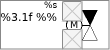
VISUALIZATION StellAntrieb_ML_Valve_Flow_LA_CheckEnabled  // 110x50
VAR_INPUT
    ITF_STELLANTRIEB_IN   	:   ITF_STELLANTRIEB;
	stExklParameter			:	STRING[40];
END_VAR
    Frame (61,0 50x50), invisible if: NOT ITF_STELLANTRIEB_IN.proIsEnabled
        shows Icon_ML_Durchfluss(ITF_STELLANTRIEB_IN := ITF_STELLANTRIEB_IN)
    Frame (0,0 60x25), invisible if: NOT ITF_STELLANTRIEB_IN.proIsEnabled
        shows ValueUpDwn(ITF_STELLANTRIEB_IN := ITF_STELLANTRIEB_IN, uiTextAusrichtung := 6)
    Rectangle (0,0 110x50)
        OnMouseClick:  Dialog=StellAntrieb_POPUP, Parameters={stExklParameter: stExklParameter, ITF_STELLANTRIEBIN: ITF_STELLANTRIEB_IN, uiPopUpGruppe: 0}, OpenCentered=True
END_VISUALIZATION

// 40 Visualizations/ICON/StellAntrieb_LEFT/Motor_LEFT/Valve_Flow/Above/StellAntrieb_ML_Valve_Flow_LA_CheckQuerry
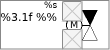
VISUALIZATION StellAntrieb_ML_Valve_Flow_LA_CheckQuerry  // 110x50
VAR_INPUT
    ITF_STELLANTRIEB_IN   	:   ITF_STELLANTRIEB;
	stExklParameter			:	STRING[40];
END_VAR
    Frame (0,0 110x50)
        shows StellAntrieb_ML_Valve_Flow_LA_CheckEnabled(ITF_STELLANTRIEB_IN := ITF_STELLANTRIEB_IN, stExklParameter := stExklParameter)
END_VISUALIZATION

// 40 Visualizations/ICON/StellAntrieb_LEFT/Motor_LEFT/Valve_Flow/Above/StellAntrieb_ML_Valve_Flow_Txt_L_Above
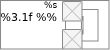
VISUALIZATION StellAntrieb_ML_Valve_Flow_Txt_L_Above  // 110x50
VAR_INPUT
    ITF_STELLANTRIEB_IN   	:   ITF_STELLANTRIEB;	
END_VAR
VAR_INPUT CONSTANT
	stExklParameter			:	STRING[40] := '';
END_VAR
VAR CONSTANT
	uiIconNr				: 	UINT := 12;
END_VAR
    Frame (0,0 110x50), invisible if: NOT fcCheckQuerryReturnIcon(_ITF_In := ITF_STELLANTRIEB_IN,_uiIconNr_In := uiIconNr)
        shows StellAntrieb_ML_Valve_Flow_LA_CheckQuerry(ITF_STELLANTRIEB_IN := ITF_STELLANTRIEB_IN, stExklParameter := stExklParameter)
        shows S_AT_ML_Valve_AB_Up_LA_CheckQuerry()
END_VISUALIZATION

// 40 Visualizations/ICON/StellAntrieb_LEFT/Motor_LEFT/Valve_Flow/Below/StellAntrieb_ML_Valve_Flow_LB_CheckEnabled
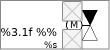
VISUALIZATION StellAntrieb_ML_Valve_Flow_LB_CheckEnabled  // 110x50
VAR_INPUT
    ITF_STELLANTRIEB_IN   	:   ITF_STELLANTRIEB;	
	stExklParameter			:	STRING[40];
END_VAR
    Frame (61,0 50x50), invisible if: NOT ITF_STELLANTRIEB_IN.proIsEnabled
        shows Icon_ML_Durchfluss(ITF_STELLANTRIEB_IN := ITF_STELLANTRIEB_IN)
    Frame (0,25 60x25), invisible if: NOT ITF_STELLANTRIEB_IN.proIsEnabled
        shows ValueDwnUp(ITF_STELLANTRIEB_IN := ITF_STELLANTRIEB_IN, uiTextAusrichtung := 6)
    Rectangle (0,0 110x50)
        OnMouseClick:  Dialog=StellAntrieb_POPUP, Parameters={stExklParameter: stExklParameter, ITF_STELLANTRIEBIN: ITF_STELLANTRIEB_IN, uiPopUpGruppe: 0}, OpenCentered=True
END_VISUALIZATION

// 40 Visualizations/ICON/StellAntrieb_LEFT/Motor_LEFT/Valve_Flow/Below/StellAntrieb_ML_Valve_Flow_LB_CheckQuerry
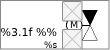
VISUALIZATION StellAntrieb_ML_Valve_Flow_LB_CheckQuerry  // 110x50
VAR_INPUT
    ITF_STELLANTRIEB_IN  	:   ITF_STELLANTRIEB;	
	stExklParameter			:	STRING[40];
END_VAR
    Frame (0,0 110x50)
        shows StellAntrieb_ML_Valve_Flow_LB_CheckEnabled(ITF_STELLANTRIEB_IN := ITF_STELLANTRIEB_IN, stExklParameter := stExklParameter)
END_VISUALIZATION

// 40 Visualizations/ICON/StellAntrieb_LEFT/Motor_LEFT/Valve_Flow/Below/StellAntrieb_ML_Valve_Flow_Txt_L_Below
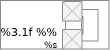
VISUALIZATION StellAntrieb_ML_Valve_Flow_Txt_L_Below  // 110x50
VAR_INPUT
    ITF_STELLANTRIEB_IN   	:   ITF_STELLANTRIEB;	
END_VAR
VAR_INPUT CONSTANT
	stExklParameter			:	STRING[40] := '';
END_VAR
VAR CONSTANT
	uiIconNr				: 	UINT := 13;
END_VAR
    Frame (0,0 110x50), invisible if: NOT fcCheckQuerryReturnIcon(_ITF_In := ITF_STELLANTRIEB_IN,_uiIconNr_In := uiIconNr)
        shows StellAntrieb_ML_Valve_Flow_LB_CheckQuerry(ITF_STELLANTRIEB_IN := ITF_STELLANTRIEB_IN, stExklParameter := stExklParameter)
        shows Icon()
END_VISUALIZATION

// 40 Visualizations/ICON/StellAntrieb_LEFT/Motor_LEFT/Valve_Mix/Above/StellAntrieb_ML_Valve_Mix_LA_CheckEnabled
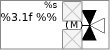
VISUALIZATION StellAntrieb_ML_Valve_Mix_LA_CheckEnabled  // 110x50
VAR_INPUT
    ITF_STELLANTRIEB_IN   	:   ITF_STELLANTRIEB;
	stExklParameter			:	STRING[40];
END_VAR
    Frame (61,0 50x50), invisible if: NOT ITF_STELLANTRIEB_IN.proIsEnabled
        shows Icon_ML_Verteiler(ITF_STELLANTRIEB_IN := ITF_STELLANTRIEB_IN)
    Frame (0,0 60x25), invisible if: NOT ITF_STELLANTRIEB_IN.proIsEnabled
        shows ValueUpDwn(ITF_STELLANTRIEB_IN := ITF_STELLANTRIEB_IN, uiTextAusrichtung := 6)
    Rectangle (0,0 110x50)
        OnMouseClick:  Dialog=StellAntrieb_POPUP, Parameters={stExklParameter: stExklParameter, ITF_STELLANTRIEBIN: ITF_STELLANTRIEB_IN, uiPopUpGruppe: 0}, OpenCentered=True
END_VISUALIZATION

// 40 Visualizations/ICON/StellAntrieb_LEFT/Motor_LEFT/Valve_Mix/Above/StellAntrieb_ML_Valve_Mix_LA_CheckQuerry
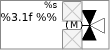
VISUALIZATION StellAntrieb_ML_Valve_Mix_LA_CheckQuerry  // 110x50
VAR_INPUT
    ITF_STELLANTRIEB_IN   	:   ITF_STELLANTRIEB;
	stExklParameter			:	STRING[40];
END_VAR
    Frame (0,0 110x50)
        shows StellAntrieb_ML_Valve_Mix_LA_CheckEnabled(ITF_STELLANTRIEB_IN := ITF_STELLANTRIEB_IN, stExklParameter := stExklParameter)
END_VISUALIZATION

// 40 Visualizations/ICON/StellAntrieb_LEFT/Motor_LEFT/Valve_Mix/Above/StellAntrieb_ML_Valve_Mix_Txt_L_Above
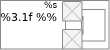
VISUALIZATION StellAntrieb_ML_Valve_Mix_Txt_L_Above  // 110x50
VAR_INPUT
    ITF_STELLANTRIEB_IN   	:   ITF_STELLANTRIEB;	
END_VAR
VAR_INPUT CONSTANT
	stExklParameter			:	STRING[40] := '';
END_VAR
VAR CONSTANT
	uiIconNr				: 	UINT := 14;
END_VAR
    Frame (0,0 110x50), invisible if: NOT fcCheckQuerryReturnIcon(_ITF_In := ITF_STELLANTRIEB_IN,_uiIconNr_In := uiIconNr)
        shows StellAntrieb_ML_Valve_Mix_LA_CheckQuerry(ITF_STELLANTRIEB_IN := ITF_STELLANTRIEB_IN, stExklParameter := stExklParameter)
        shows S_AT_ML_Valve_AB_Up_LA_CheckQuerry()
END_VISUALIZATION

// 40 Visualizations/ICON/StellAntrieb_LEFT/Motor_LEFT/Valve_Mix/Below/StellAntrieb_ML_Valve_Mix_LB_CheckEnabled
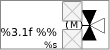
VISUALIZATION StellAntrieb_ML_Valve_Mix_LB_CheckEnabled  // 110x50
VAR_INPUT
    ITF_STELLANTRIEB_IN   	:   ITF_STELLANTRIEB;
	stExklParameter			:	STRING[40];
END_VAR
    Frame (61,0 50x50), invisible if: NOT ITF_STELLANTRIEB_IN.proIsEnabled
        shows Icon_ML_Verteiler(ITF_STELLANTRIEB_IN := ITF_STELLANTRIEB_IN)
    Frame (0,25 60x25), invisible if: NOT ITF_STELLANTRIEB_IN.proIsEnabled
        shows ValueDwnUp(ITF_STELLANTRIEB_IN := ITF_STELLANTRIEB_IN, uiTextAusrichtung := 6)
    Rectangle (0,0 110x50)
        OnMouseClick:  Dialog=StellAntrieb_POPUP, Parameters={stExklParameter: stExklParameter, ITF_STELLANTRIEBIN: ITF_STELLANTRIEB_IN, uiPopUpGruppe: 0}, OpenCentered=True
END_VISUALIZATION

// 40 Visualizations/ICON/StellAntrieb_LEFT/Motor_LEFT/Valve_Mix/Below/StellAntrieb_ML_Valve_Mix_LB_CheckQuerry
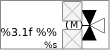
VISUALIZATION StellAntrieb_ML_Valve_Mix_LB_CheckQuerry  // 110x50
VAR_INPUT
    ITF_STELLANTRIEB_IN   	:   ITF_STELLANTRIEB;
	stExklParameter			:	STRING[40];
END_VAR
    Frame (0,0 110x50)
        shows StellAntrieb_ML_Valve_Mix_LB_CheckEnabled(ITF_STELLANTRIEB_IN := ITF_STELLANTRIEB_IN, stExklParameter := stExklParameter)
END_VISUALIZATION

// 40 Visualizations/ICON/StellAntrieb_LEFT/Motor_LEFT/Valve_Mix/Below/StellAntrieb_ML_Valve_Mix_Txt_L_Below
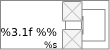
VISUALIZATION StellAntrieb_ML_Valve_Mix_Txt_L_Below  // 110x50
VAR_INPUT
    ITF_STELLANTRIEB_IN   	:   ITF_STELLANTRIEB;	
END_VAR
VAR_INPUT CONSTANT
	stExklParameter			:	STRING[40] := '';
END_VAR
VAR CONSTANT
	uiIconNr				: 	UINT := 15;
END_VAR
    Frame (0,0 110x50), invisible if: NOT fcCheckQuerryReturnIcon(_ITF_In := ITF_STELLANTRIEB_IN,_uiIconNr_In := uiIconNr)
        shows StellAntrieb_ML_Valve_Mix_LB_CheckQuerry(ITF_STELLANTRIEB_IN := ITF_STELLANTRIEB_IN, stExklParameter := stExklParameter)
        shows Icon()
END_VISUALIZATION

// 40 Visualizations/POPUP/PARAMETER/StellAntrieb_Icon_StellAntrieb
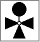
VISUALIZATION StellAntrieb_Icon_StellAntrieb  // 40x42
    Group (5,2 28x36)
        Ellipse (7,0 14x14)
        Polygon (0,15) (14,21) (0,27)
        Polygon (14,22) (20,36) (8,36)
        Polygon (14,21) (28,15) (28,27)
        Line (14,21) (14,14)
        Ellipse (12,19 4x4)
END_VISUALIZATION

// 40 Visualizations/POPUP/PARAMETER/StellAntrieb_POPUP_IO_ITF
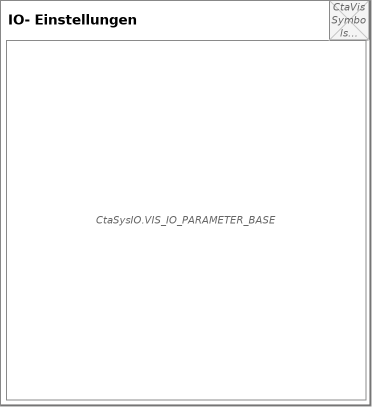
VISUALIZATION StellAntrieb_POPUP_IO_ITF  // 372x407
VAR_INPUT
    ITF_IO_IN    :   CtaSysIO.ITF_IO;	
END_VAR
    RoundedRectangle (0,0 370x405)
    Frame (6,40 360x360)
        shows CtaSysIO.VIS_IO_PARAMETER_BASE(ITF_IO_IN := ITF_IO_IN)
        shows VIS_ANTRIEB_PARAMETER_IO1(ITF_ANTRIEBIN := ITF_ANTRIEBIN)
        shows VIS_ANTRIEB_PARAMETER_IO2(ITF_ANTRIEBIN := ITF_ANTRIEBIN)
        shows VIS_ANTRIEB_PARAMETER_IO3(ITF_ANTRIEBIN := ITF_ANTRIEBIN)
    Image (329,0 40x40), image: CtaVisSymbols.ImagePool.close_solo_black
        OnMouseClick:  Dialog=StellAntrieb_POPUP_IO_ITF, Result=None, NumpadKeypadSet=True
    Label (5,0 150x40), "IO- Einstellungen"
END_VISUALIZATION

// 40 Visualizations/POPUP/PARAMETER/StellAntrieb_IO/StellAntrieb_ParameterIO4
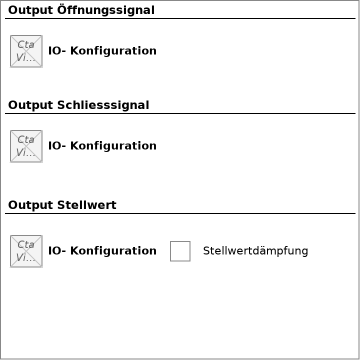
VISUALIZATION StellAntrieb_ParameterIO4  // 360x360
VAR_INPUT
    ITF_STELLANTRIEBIN  :   ITF_STELLANTRIEB;	
	ITF_xOnAuf_IN		:	CtaSysIO.ITF_IO;
	ITF_xOnZu_IN		:	CtaSysIO.ITF_IO;
	ITF_rOnY_IN			:	CtaSysIO.ITF_IO;
END_VAR
    Label (5,0 350x20), "Output Öffnungssignal"
    Label (5,195 350x20), "Output Stellwert"
    Line (5,213) (355,213)
    Line (5,18) (355,18)
    Image (10,35 32x32), invisible if: ITF_xOnAuf_IN = 0, image: CtaVisSymbols.ImagePool.build
        OnMouseDown:  Dialog=StellAntrieb_POPUP_IO_ITF, Parameters={ITF_IO_IN: ITF_xOnAuf_IN}, OpenModal=True, OpenCentered=True
    Image (10,235 32x32), invisible if: ITF_rOnY_IN = 0, image: CtaVisSymbols.ImagePool.build
        OnMouseDown:  Dialog=StellAntrieb_POPUP_IO_ITF, Parameters={ITF_IO_IN: ITF_rOnY_IN}, OpenModal=True, OpenCentered=True
    Label (45,41 120x20), "IO- Konfiguration", invisible if: ITF_xOnAuf_IN = 0
    Label (45,241 120x20), "IO- Konfiguration", invisible if: ITF_rOnY_IN = 0
    Line (5,113) (355,113)
    Label (5,95 350x20), "Output Schliesssignal"
    Image (10,130 32x32), invisible if: ITF_xOnZu_IN = 0, image: CtaVisSymbols.ImagePool.build
        OnMouseDown:  Dialog=StellAntrieb_POPUP_IO_ITF, Parameters={ITF_IO_IN: ITF_xOnZu_IN}, OpenModal=True, OpenCentered=True
    Label (45,136 120x20), "IO- Konfiguration", invisible if: ITF_xOnZu_IN = 0
    Label (200,241 150x20), "Stellwertdämpfung"
    Frame (170,241 20x20)
        shows CtaAppDumper.VisDumperSmall(fbDumper := ITF_STELLANTRIEBIN.proRefToRonYDumper)
END_VISUALIZATION

// 40 Visualizations/POPUP/PARAMETER/StellAntrieb_ParameterBase/StellAntrieb_ParameterBase2
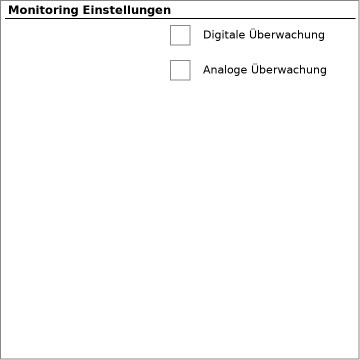
VISUALIZATION StellAntrieb_ParameterBase2  // 360x360
VAR_INPUT
    ITF_STELLANTRIEBIN : ITF_STELLANTRIEB;
END_VAR
    Label (5,0 350x20), "Monitoring Einstellungen"
    Frame (170,25 20x20)
        shows CtaSysConfig.visBOOL(visfbBOOLIn := ITF_STELLANTRIEBIN.p_scBase_fbxEnDigitalMonitoring)
    Label (200,25 150x20), "Digitale Überwachung"
    Frame (170,60 20x20)
        shows CtaSysConfig.visBOOL(visfbBOOLIn := ITF_STELLANTRIEBIN.p_scBase_fbxEnAnalogMonitoring)
    Label (200,60 150x20), "Analoge Überwachung"
    Line (5,18) (355,18)
END_VISUALIZATION

// 40 Visualizations/POPUP/PARAMETER/StellAntrieb_ParameterBase/StellAntrieb_ParameterBase1
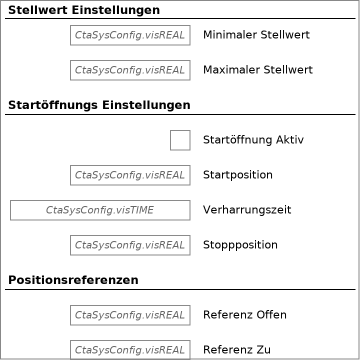
VISUALIZATION StellAntrieb_ParameterBase1  // 360x360
VAR_INPUT
    ITF_STELLANTRIEBIN : ITF_STELLANTRIEB;
END_VAR
    Label (5,0 350x20), "Stellwert Einstellungen"
    Frame (70,25 120x20)
        shows CtaSysConfig.visREAL(visfbREALIn := ITF_STELLANTRIEBIN.p_scBase_fbrYMin, stPhysikalischeEinheit := '%')
    Label (200,25 150x20), "Minimaler Stellwert"
    Label (200,60 150x20), "Maximaler Stellwert"
    Frame (70,60 120x20)
        shows CtaSysConfig.visREAL(visfbREALIn := ITF_STELLANTRIEBIN.p_scBase_fbrYMax, stPhysikalischeEinheit := '%')
    Frame (170,130 20x20)
        shows CtaSysConfig.visBOOL(visfbBOOLIn := ITF_STELLANTRIEBIN.p_scBase_fbxEnStartPosition)
    Label (200,130 150x20), "Startöffnung Aktiv"
    Frame (70,165 120x20)
        shows CtaSysConfig.visREAL(visfbREALIn := ITF_STELLANTRIEBIN.p_scBase_fbrYStartPos, stPhysikalischeEinheit := '%')
    Label (200,165 150x20), "Startposition"
    Frame (10,200 180x20)
        shows CtaSysConfig.visTIME(visfbTIMEIn := ITF_STELLANTRIEBIN.p_scBase_fbtStartPosTime)
    Label (200,200 150x20), "Verharrungszeit"
    Frame (70,235 120x20)
        shows CtaSysConfig.visREAL(visfbREALIn := ITF_STELLANTRIEBIN.p_scBase_fbrYStopp, stPhysikalischeEinheit := '%')
    Label (200,235 150x20), "Stoppposition"
    Label (200,305 150x20), "Referenz Offen"
    Frame (70,305 120x20)
        shows CtaSysConfig.visREAL(visfbREALIn := ITF_STELLANTRIEBIN.p_scBase_fbrRefIsOpen, stPhysikalischeEinheit := '%')
    Label (200,340 150x20), "Referenz Zu"
    Frame (70,340 120x20)
        shows CtaSysConfig.visREAL(visfbREALIn := ITF_STELLANTRIEBIN.p_scBase_fbrRefIsClosed, stPhysikalischeEinheit := '%')
    Label (5,95 350x20), "Startöffnungs Einstellungen"
    Label (5,270 350x20), "Positionsreferenzen"
    Line (5,18) (355,18)
    Line (5,114) (355,114)
    Line (5,289) (355,289)
END_VISUALIZATION

// 40 Visualizations/ICON/StellAntrieb_BASE/Value/ValueUpDwn
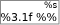
VISUALIZATION ValueUpDwn  // 60x25
VAR_INPUT
    ITF_STELLANTRIEB_IN   :   ITF_STELLANTRIEB;	
END_VAR
VAR_INPUT CONSTANT
    uiTextAusrichtung   : UINT := 4;    // 0 = Oben links | 1 = Horizontal zentriert | 2 = Rechts | 4 = Vertikal zentriert | 8 = Unten
END_VAR
    Textfield (0,0 60x10), "%s", text variable: ITF_STELLANTRIEB_IN.proGetBMK, invisible if: ITF_STELLANTRIEB_IN.proNoBmkInList
        p3718999670: uiTextAusrichtung
    Textfield (0,10 60x15), "%3.1f %%", text variable: ITF_STELLANTRIEB_IN.proOnY, invisible if: NOT ITF_STELLANTRIEB_IN.proIsRegulatet
        p3718999670: uiTextAusrichtung
END_VISUALIZATION

// 40 Visualizations/ICON/StellAntrieb_BASE/Value/ValueDwnUp
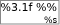
VISUALIZATION ValueDwnUp  // 60x25
VAR_INPUT
    ITF_STELLANTRIEB_IN   :   ITF_STELLANTRIEB;	
END_VAR
VAR_INPUT CONSTANT
    uiTextAusrichtung   : UINT := 4;    // 0 = Oben links | 1 = Horizontal zentriert | 2 = Rechts | 4 = Vertikal zentriert | 8 = Unten
END_VAR
    Textfield (0,0 60x15), "%3.1f %%", text variable: ITF_STELLANTRIEB_IN.proOnY, invisible if: NOT ITF_STELLANTRIEB_IN.proIsRegulatet
        p3718999670: uiTextAusrichtung
    Textfield (0,15 60x10), "%s", text variable: ITF_STELLANTRIEB_IN.proGetBMK, invisible if: ITF_STELLANTRIEB_IN.proNoBmkInList
        p3718999670: uiTextAusrichtung
END_VISUALIZATION

(* text list Error (id | default | de | en | fr | it)
  0 | keine Meldung Anstehend | Keine Meldung Anstehend | No message pending | Aucun message en attente | Nessun messaggio in sospeso
  1 | Die Abweichung des Stellwertes zum Istwert ist zu hoch | Die Abweichung des Stellwertes zum Istwert ist zu hoch | The deviation of the control value from the actual value is too high /  | L'écart entre la valeur de contrôle et la valeur réelle est trop élevé | Lo scostamento del valore di controllo dal valore effettivo è troppo elevato
  3 | Keine Rückmeldung des Stellventils beim öffnen | Keine Rückmeldung des Stellventils beim öffnen | No feedback from the control valve when opening | Pas de retour de la vanne de régulation lors de l'ouverture | Nessun feedback dalla valvola di controllo durante l'apertura
  2 | Keine Rückmeldung des Stellventils beim schlissen | Keine Rückmeldung des Stellventils beim schlissen | No feedback from the control valve when closing | Pas de retour de la vanne de régulation lors de la fermeture | Nessun feedback dalla valvola di controllo durante la chiusura
  4 | Digitaler Stellwert nicht erreicht | Digitaler Stellwert nicht erreicht | Digital control value not reached | Valeur de contrôle numérique non atteinte | Valore di controllo digitale non raggiunto
  5 | Analoger Stellwert nicht erreicht | Analoger Stellwert nicht erreicht | Analog control value not reached | Valeur de contrôle analogique non atteinte | Valore di controllo analogico non raggiunto
  6 | Leitungsschutzschalter ausfall | Leitungsschutzschalter ausfall | Circuit breaker failure | Défaillance du disjoncteur | Guasto dell'interruttore
  7 | Motorschutzschalter ausfall | Motorschutzschalter ausfall | Motor protection switch failure | Défaillance de l'interrupteur de protection du moteur | Guasto al salvamotore
  8 | Konfigurationsfehler speichern fehlgeschlagen reboot | Konfigurationsfehler speichern fehlgeschlagen reboot | Failed to save configuration error reboot | Impossible d'enregistrer l'erreur de configuration reboot | Impossibile salvare l'errore di configurazione reboot
   |  |  |  |  |  *)

(* text list Info (id | default | de | en | fr | it)
  0 | keine Meldung Anstehend | keine Meldung Anstehend | no message pending | aucun message en attente | nessun messaggio in sospeso
   |  |  |  |  |  *)

(* text list Warnung (id | default | de | en | fr | it)
  0 | Keine Meldung Anstehend | Keine Meldung Anstehend | No message pending | Aucun message en attente | Nessun messaggio in sospeso
  3 | Wahlschalter Hand, Ein | Wahlschalter Hand, Ein | Selector switch hand on | Commutateur de sélection a main, Allumé | Selettore a mano, acceso
  2 | Wahlschalter Hand, Aus | Wahlschalter Hand, Aus | Selector switch hand off | Commutateur de sélection a main, Éteint | Selettore a mano, spento
  1 | Revisionsschalter Ausgeschalten | Revisionsschalter Ausgeschalten | Revision switch off | Commutateur révision Désactiver | Interruttore di revisione disattivato
  4 | Handmodul aktiv | Handmodul aktiv | Hand module active | Module manuel actif | Modulo manuale attivo
   |  |  |  |  |  *)
